(* CODESYS project CFC_R_TRIG.xml

Project tree, tasks and I/O mapping:
  function CFC_R_TRIG [CFC]
*)

// CFC_R_TRIG
FUNCTION CFC_R_TRIG : BOOL
VAR_INPUT
	CLK : BOOL;
END_VAR


VAR_IN_OUT
	aux_mem : BOOL;
END_VAR

VAR_OUTPUT
	Q : BOOL;
END_VAR

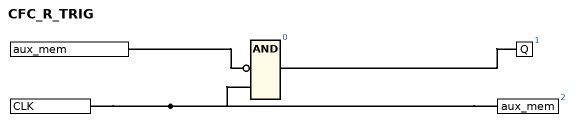
Q := NOT aux_mem AND CLK;
aux_mem := CLK;

END_FUNCTION
